FUNCTION FUN_Scale : REAL
VAR_INPUT
	ix : REAL;
	ixmax : REAL;
	ixmin : REAL;
	rymax : REAL;
	rymin : REAL;
END_VAR
VAR
	rk : REAL := 0.085449218;
	rd : REAL := 0;
END_VAR

rk := (rymax - rymin) / (ixmax - ixmin);
rd := rymin - rk * ixmin;

FUN_Scale := rk * ix +rd;

IF FUN_Scale > rymax THEN
	FUN_Scale := rymax;
ELSIF FUN_Scale < rymin THEN
	FUN_Scale := rymin;
END_IF

END_FUNCTION

(* stored: Version 1.1.0.1, ProductVersion 3.1.4024.15
   POU FUN_Scale: Id {b2ad5e09-a1d4-4cd7-aad6-fef559f2c9c5}, SpecialFunc None *)
